{attribute addProperty BoxType "EJ7411-0000-0018"}
{attribute addProperty Id "Target_positionAT %Q*UDINT324"}
{attribute addProperty CRC "1093881770"}
{attribute addProperty SizeInBites "32"}
{attribute addProperty SizeInBytes "4"}
TYPE DRV_Target_position_41334FAA :
STRUCT
	{attribute addProperty Name "Target_position"}
	Target_position AT %Q* : UDINT;
END_STRUCT
END_TYPE

(* stored: Version 1.2.0.0, ProductVersion 3.1.4024.9
   DUT DRV_Target_position_41334FAA: Id {1f0c53e1-b6a1-4949-aff0-21546a6e9303} *)
